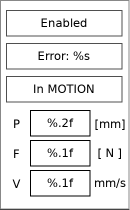
VISUALIZATION vHP3_AxisMainParamsDisplay  // 130x210
VAR_IN_OUT
	fbAxis	: fbHP_Axis;
END_VAR
    RoundedRectangle (0,0 129x210)
    Rectangle (30,110 60x26), "%.2f", text variable: fbAxis.McReadActualPosition.Position
    Label (93,111 34x26), "[mm]"
    Label (4,111 25x26), "P"
    Rectangle (30,140 60x26), "%.1f", text variable: fbAxis.fbForceFilter.rOut
    Label (93,140 34x26), "[ N ]"
    Label (4,141 25x26), "F"
    Rectangle (30,170 60x26), "%.1f", text variable: fbAxis.McReadActualVelocity.ActualVelocity, colour toggle: fbAxis.IsMoving
    Label (93,170 34x26), "mm/s"
    Label (4,171 25x26), "V"
    Rectangle (6,43 116x26), "Error: %s", text variable: TO_STRING(fbAxis.nActEvent), colour toggle: fbAxis.IsErrorActive
    Rectangle (6,10 116x26), "Enabled", colour toggle: fbAxis.Enabled
    Rectangle (6,76 116x26), "In MOTION", text variable: TO_STRING(fbAxis.nActEvent), colour toggle: fbAxis.IsMoving
END_VISUALIZATION

(* stored: Version 1.1.0.1, ProductVersion 3.1.4024.12
   Visu vHP3_AxisMainParamsDisplay: Id {0e0c2b3f-75f9-470e-b952-4a048c1f7ed4} *)
